(* IEC 61131-3 sources: test/Class/_LseEasyLanguage, 1 file *)

(* ---- _LseEasyLanguage.st ---- *)
(*!
<Class
	Name               = "_LseEasyLanguage"
	Revision           = "1.0"
	RealtimeTask       = "false"
	CyclicTask         = "false"
	BackgroundTask     = "false"
	Sigmatek           = "true"
	OSInterface        = "false"
	HighPriority       = "false"
	Automatic          = "false"
	UpdateMode         = "Prescan"
	SharedCommandTable = "true"
	Objectsize         = "(480,120)"
	Comment            = "Language Selection for Lse Easy&#13;&#10;Writes the selected language via object channel to the LseEasy object.">
	<Channels>
		<Server Name="SelLanguageBit" Visualized="true" Initialize="false" WriteProtected="false" Retentive="File" Comment="Server for BITWISE language selection. &#13;&#10;Bit 0: select language 1 of the &quot;Languages to compile&quot; list of LSE project&#13;&#10;Bit 1: select language 2 of the &quot;Languages to compile&quot; list of LSE project&#13;&#10;Bit 2: select language 3 of the &quot;Languages to compile&quot; list of LSE project&#13;&#10;and so on ...&#13;&#10;"/>
		<Client Name="_Radio321" Required="true" Internal="true"/>
		<Client Name="LseEasy" Required="true" Internal="false" Comment="object channel to the LseEasy object"/>
	</Channels>
	<RevDoku>
		<Owner Company="Sigmatek GmbH" Author="Weitho"/>
		<Dokumentation Revision="1.0" Date="2017-05-03" Author="KaiAnd" Company="Sigmatek GmbH" Description="Creation of class"/>
	</RevDoku>
	<Network Name="_LseEasyLanguage">
		<!-- List of Components in this network -->
		<Components>
			<Object
				Name       = "_Radio321"
				Class      = "_Radio32"
				Position   = "(180,180)"
				Visualized = "true"
				Remotely   = "true">
				<Channels>
					<Server Name="Data"/>
				</Channels>
			</Object>
		</Components>
		<Comments>
		</Comments>
		<!-- List of Connections in this network -->
		<Connections>
			<Connection Source="this._Radio321" Destination="_Radio321.Data"/>
		</Connections>
		<!-- Headerfiles -->
		<Options>
		</Options>
	</Network>
</Class>
*)
_LseEasyLanguage : CLASS
	TYPE
	  TYPE_Language : BDINT  //! <Type Public="true" Name="TYPE_Language"/>
	  [
	    1 L_DE,
	    2 L_GB,
	  ];
	END_TYPE
  //Servers:
	SelLanguageBit 	: SvrChCmd_TYPE_Language_PTofCls__LseEasyLanguage;
  //Clients:
	LseEasy 	: CltChCmd_LseEasy;
	_Radio321 	: CltChCmd__Radio32;
  //Variables:
  //Functions:

	FUNCTION VIRTUAL GLOBAL Init;

	FUNCTION VIRTUAL GLOBAL SelLanguageBit::Write
		VAR_INPUT
			input (EAX) 	: _LseEasyLanguage::TYPE_Language;
		END_VAR
		VAR_OUTPUT
			result (EAX) 	: _LseEasyLanguage::TYPE_Language;
		END_VAR;
  //Tables:
	FUNCTION @STD
		VAR_OUTPUT
			ret_code	: CONFSTATES;
		END_VAR;
	FUNCTION GLOBAL TAB @CT_;
END_CLASS;

#pragma using _Radio32
#pragma usingLtd LseEasy

FUNCTION VIRTUAL GLOBAL _LseEasyLanguage::Init

  if (_FirstScan) then

    if (SelLanguageBit = 0) then
      SelLanguageBit := 1;
    end_if;

  end_if;

END_FUNCTION

FUNCTION VIRTUAL GLOBAL _LseEasyLanguage::SelLanguageBit::Write
	VAR_INPUT
		input (EAX) 	: _LseEasyLanguage::TYPE_Language;
	END_VAR
	VAR_OUTPUT
		result (EAX) 	: _LseEasyLanguage::TYPE_Language;
	END_VAR
  VAR
	  LangIdx  : UDINT;
    myBit    : BDINT;
    u        : UDINT;
  END_VAR

	SelLanguageBit := _Radio321.Data.Write(input:=input);
	result := SelLanguageBit;

  myBit   := SelLanguageBit;
  LangIdx := 0;   // Index in "Languages to compile" list of LSE project

  // convert  Bit-Nr. to index (0-31)
  for u:=0 to 31 do

    if ( (myBit SHR u) and 1) then
      LangIdx := u;
      exit;
    end_if;

  end_for;

  LseEasy.ActLanguage.Write(LangIdx);

END_FUNCTION
